// Mitsubishi GX Works2 project: geothermal   PLC: FX3U/FX3UC

PROGRAM MAIN
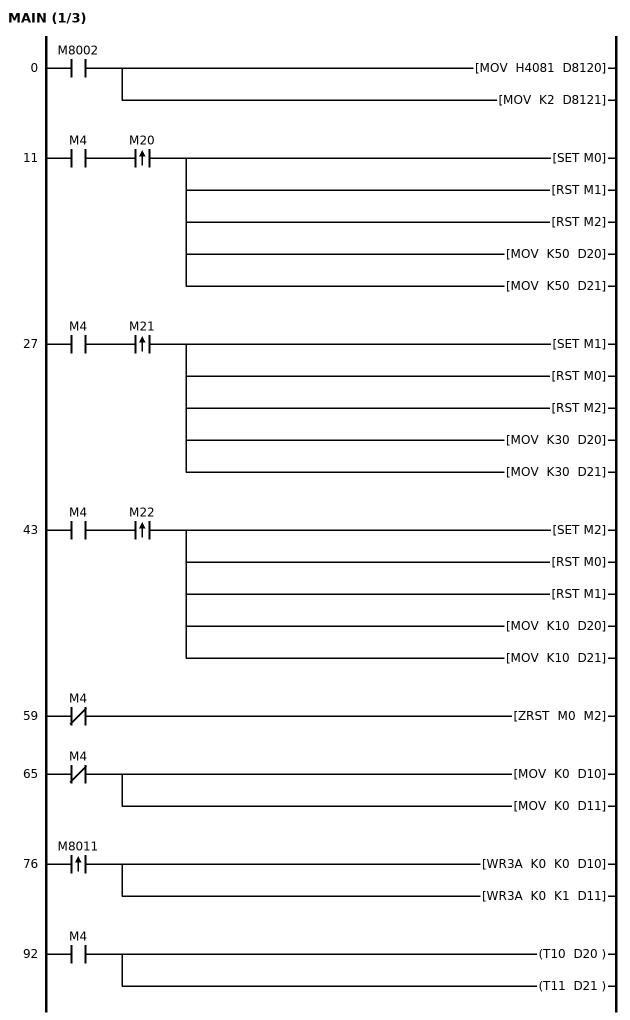
0     LD      M8002
      MOV     H4081 D8120
      MOV     K2 D8121
11    LD      M4
      ANDP    M20
      SET     M0
      RST     M1
      RST     M2
      MOV     K50 D20
      MOV     K50 D21
27    LD      M4
      ANDP    M21
      SET     M1
      RST     M0
      RST     M2
      MOV     K30 D20
      MOV     K30 D21
43    LD      M4
      ANDP    M22
      SET     M2
      RST     M0
      RST     M1
      MOV     K10 D20
      MOV     K10 D21
59    LDI     M4
      ZRST    M0 M2
65    LDI     M4
      MOV     K0 D10
      MOV     K0 D11
76    LDP     M8011
      WR3A    K0 K0 D10
      WR3A    K0 K1 D11
92    LD      M4
      OUT     T10 D20
      OUT     T11 D21
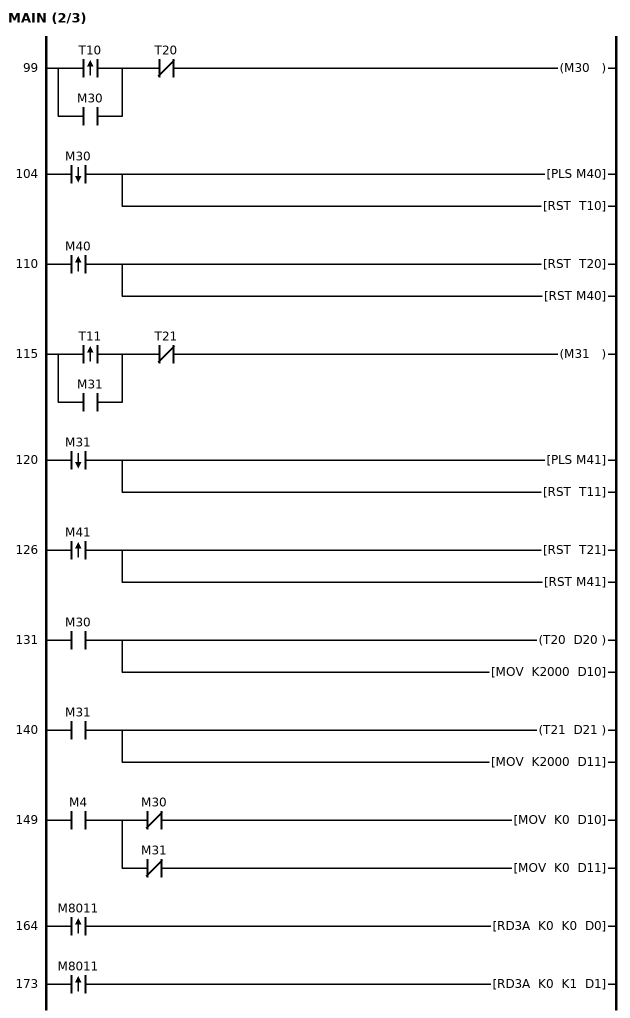
99    LDP     T10
      OR      M30
      ANI     T20
      OUT     M30
104   LDF     M30
      PLS     M40
      RST     T10
110   LDP     M40
      RST     T20
      RST     M40
115   LDP     T11
      OR      M31
      ANI     T21
      OUT     M31
120   LDF     M31
      PLS     M41
      RST     T11
126   LDP     M41
      RST     T21
      RST     M41
131   LD      M30
      OUT     T20 D20
      MOV     K2000 D10
140   LD      M31
      OUT     T21 D21
      MOV     K2000 D11
149   LD      M4
      MPS
      ANI     M30
      MOV     K0 D10
      MPP
      ANI     M31
      MOV     K0 D11
164   LDP     M8011
      RD3A    K0 K0 D0
173   LDP     M8011
      RD3A    K0 K1 D1
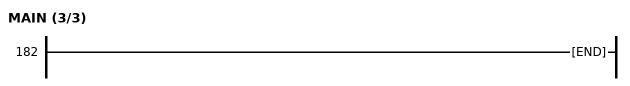
182   END
END_PROGRAM
